// TIA Portal V17 export
// export: Created 2022-06-27T13:58:12.5264541Z, ExportSetting WithDefaults, DisplayName Totally Integrated Automation Portal, DisplayVersion V17 Update 3, DisplayName TIA Portal Openness, DisplayVersion V17 Update 3, DisplayName TIA Portal Version Control Interface, DisplayVersion V17, DisplayName SINAMICS Startdrive Advanced, DisplayVersion V17 Update1, DisplayName SINAMICS Startdrive G110M, G120, G120C, G120D, G120P, G115D, DisplayVersion V17 Update1, DisplayName SINAMICS Startdrive G130, G150, S120, S150, SINAMICS MV, S210, DisplayVersion V17 Update1, DisplayName STEP 7 Professional, DisplayVersion V17 Update 3, DisplayName STEP 7 Safety, DisplayVersion V17, DisplayName WinCC UA Professional, DisplayVersion V17 Update 3
FUNCTION_BLOCK "S05_ANALOGIC_INPUTS"   // FB5, LAD
{ S7_Optimized_Access := 'TRUE' }
VERSION : 0.1
// stored: AutoNumber false, IsIECCheckEnabled false, IsRetainMemResEnabled false, MemoryReserve 100, SetENOAutomatically false, UDAEnableTagReadback false
   VAR
      FB_ANALOGIC_INPUTS_TT82_2E { S7_SetPoint := 'True'} : "FB_ANALOGIC_INPUTS";
      FB_ANALOGIC_INPUTS_TT82_4E { S7_SetPoint := 'True'} : "FB_ANALOGIC_INPUTS";
      FB_ANALOGIC_INPUTS_TT82_6E { S7_SetPoint := 'True'} : "FB_ANALOGIC_INPUTS";
      FB_ANALOGIC_INPUTS_TT82_8E { S7_SetPoint := 'True'} : "FB_ANALOGIC_INPUTS";
      FB_ANALOGIC_INPUTS_TT83_2E { S7_SetPoint := 'True'} : "FB_ANALOGIC_INPUTS";
      FB_ANALOGIC_INPUTS_TT83_4E { S7_SetPoint := 'True'} : "FB_ANALOGIC_INPUTS";
      FB_ANALOGIC_INPUTS_TT83_6E { S7_SetPoint := 'True'} : "FB_ANALOGIC_INPUTS";
      FB_ANALOGIC_INPUTS_TT88_2E { S7_SetPoint := 'True'} : "FB_ANALOGIC_INPUTS";
      FB_ANALOGIC_INPUTS_TT83_8E { S7_SetPoint := 'True'} : "FB_ANALOGIC_INPUTS";
      FB_ANALOGIC_INPUTS_TT84_4E { S7_SetPoint := 'True'} : "FB_ANALOGIC_INPUTS";
      FB_ANALOGIC_INPUTS_TT84_6E { S7_SetPoint := 'True'} : "FB_ANALOGIC_INPUTS";
      FB_ANALOGIC_INPUTS_TT84_8E { S7_SetPoint := 'True'} : "FB_ANALOGIC_INPUTS";
      FB_ANALOGIC_INPUTS_TT85_2E { S7_SetPoint := 'True'} : "FB_ANALOGIC_INPUTS";
   END_VAR
BEGIN

REGION Network 1: TT82-2E - Furnace Thermocouple
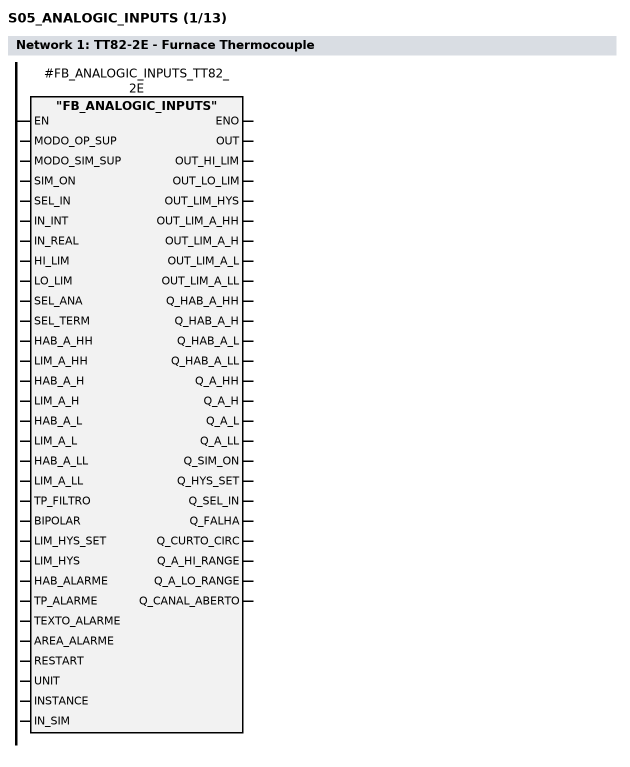
   RUNG wire#powerrail
      #FB_ANALOGIC_INPUTS_TT82_2E(MODO_OP_SUP :=, MODO_SIM_SUP :=, SIM_ON :=, SEL_IN :=, IN_INT :=, IN_REAL :=, HI_LIM :=, LO_LIM :=, SEL_ANA :=, SEL_TERM :=, HAB_A_HH :=, LIM_A_HH :=, HAB_A_H :=, LIM_A_H :=, HAB_A_L :=, LIM_A_L :=, HAB_A_LL :=, LIM_A_LL :=, TP_FILTRO :=, BIPOLAR :=, LIM_HYS_SET :=, LIM_HYS :=, HAB_ALARME :=, TP_ALARME :=, TEXTO_ALARME :=, AREA_ALARME :=, RESTART :=, UNIT :=, INSTANCE :=, IN_SIM :=, OUT =>, OUT_HI_LIM =>, OUT_LO_LIM =>, OUT_LIM_HYS =>, OUT_LIM_A_HH =>, OUT_LIM_A_H =>, OUT_LIM_A_L =>, OUT_LIM_A_LL =>, Q_HAB_A_HH =>, Q_HAB_A_H =>, Q_HAB_A_L =>, Q_HAB_A_LL =>, Q_A_HH =>, Q_A_H =>, Q_A_L =>, Q_A_LL =>, Q_SIM_ON =>, Q_HYS_SET =>, Q_SEL_IN =>, Q_FALHA =>, Q_CURTO_CIRC =>, Q_A_HI_RANGE =>, Q_A_LO_RANGE =>, Q_CANAL_ABERTO =>)
   END_RUNG
   // the same network as SCL:
   #FB_ANALOGIC_INPUTS_TT82_2E();   // "FB_ANALOGIC_INPUTS"
END_REGION

REGION Network 3: TT82-4E - Chamber 1 Air Intake Thermocouple
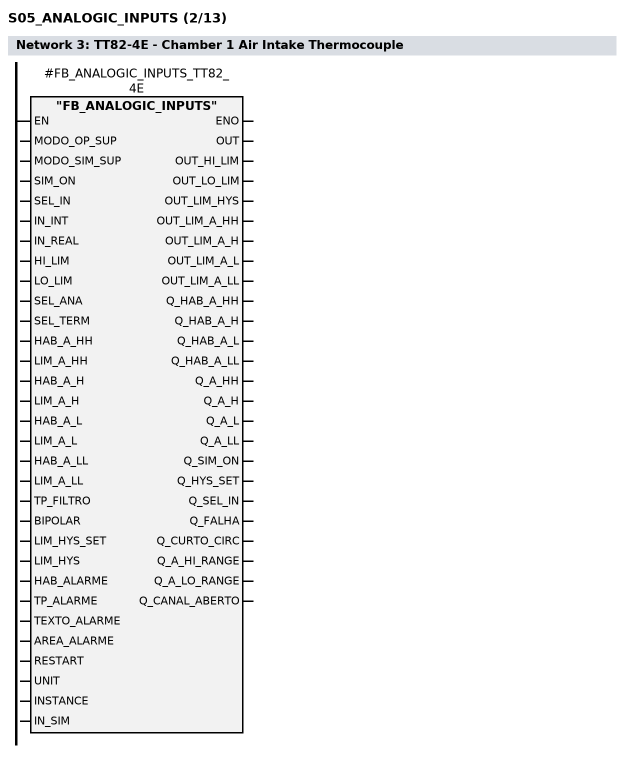
   RUNG wire#powerrail
      #FB_ANALOGIC_INPUTS_TT82_4E(MODO_OP_SUP :=, MODO_SIM_SUP :=, SIM_ON :=, SEL_IN :=, IN_INT :=, IN_REAL :=, HI_LIM :=, LO_LIM :=, SEL_ANA :=, SEL_TERM :=, HAB_A_HH :=, LIM_A_HH :=, HAB_A_H :=, LIM_A_H :=, HAB_A_L :=, LIM_A_L :=, HAB_A_LL :=, LIM_A_LL :=, TP_FILTRO :=, BIPOLAR :=, LIM_HYS_SET :=, LIM_HYS :=, HAB_ALARME :=, TP_ALARME :=, TEXTO_ALARME :=, AREA_ALARME :=, RESTART :=, UNIT :=, INSTANCE :=, IN_SIM :=, OUT =>, OUT_HI_LIM =>, OUT_LO_LIM =>, OUT_LIM_HYS =>, OUT_LIM_A_HH =>, OUT_LIM_A_H =>, OUT_LIM_A_L =>, OUT_LIM_A_LL =>, Q_HAB_A_HH =>, Q_HAB_A_H =>, Q_HAB_A_L =>, Q_HAB_A_LL =>, Q_A_HH =>, Q_A_H =>, Q_A_L =>, Q_A_LL =>, Q_SIM_ON =>, Q_HYS_SET =>, Q_SEL_IN =>, Q_FALHA =>, Q_CURTO_CIRC =>, Q_A_HI_RANGE =>, Q_A_LO_RANGE =>, Q_CANAL_ABERTO =>)
   END_RUNG
   // the same network as SCL:
   #FB_ANALOGIC_INPUTS_TT82_4E();   // "FB_ANALOGIC_INPUTS"
END_REGION

REGION Network 5: TT82-6E - Chamber 2 Air Intake Thermocouple
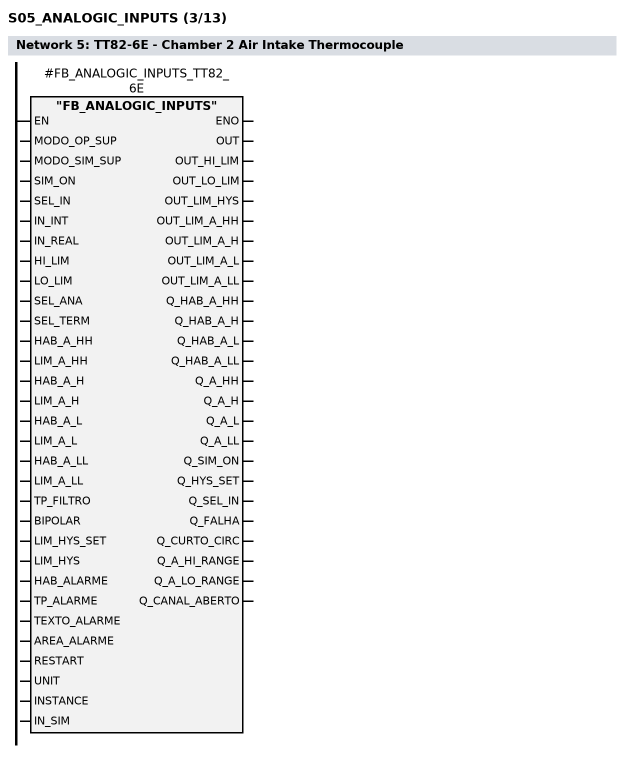
   RUNG wire#powerrail
      #FB_ANALOGIC_INPUTS_TT82_6E(MODO_OP_SUP :=, MODO_SIM_SUP :=, SIM_ON :=, SEL_IN :=, IN_INT :=, IN_REAL :=, HI_LIM :=, LO_LIM :=, SEL_ANA :=, SEL_TERM :=, HAB_A_HH :=, LIM_A_HH :=, HAB_A_H :=, LIM_A_H :=, HAB_A_L :=, LIM_A_L :=, HAB_A_LL :=, LIM_A_LL :=, TP_FILTRO :=, BIPOLAR :=, LIM_HYS_SET :=, LIM_HYS :=, HAB_ALARME :=, TP_ALARME :=, TEXTO_ALARME :=, AREA_ALARME :=, RESTART :=, UNIT :=, INSTANCE :=, IN_SIM :=, OUT =>, OUT_HI_LIM =>, OUT_LO_LIM =>, OUT_LIM_HYS =>, OUT_LIM_A_HH =>, OUT_LIM_A_H =>, OUT_LIM_A_L =>, OUT_LIM_A_LL =>, Q_HAB_A_HH =>, Q_HAB_A_H =>, Q_HAB_A_L =>, Q_HAB_A_LL =>, Q_A_HH =>, Q_A_H =>, Q_A_L =>, Q_A_LL =>, Q_SIM_ON =>, Q_HYS_SET =>, Q_SEL_IN =>, Q_FALHA =>, Q_CURTO_CIRC =>, Q_A_HI_RANGE =>, Q_A_LO_RANGE =>, Q_CANAL_ABERTO =>)
   END_RUNG
   // the same network as SCL:
   #FB_ANALOGIC_INPUTS_TT82_6E();   // "FB_ANALOGIC_INPUTS"
END_REGION

REGION Network 7: TT82-8E - Roaster Air Outtake Thermocouple
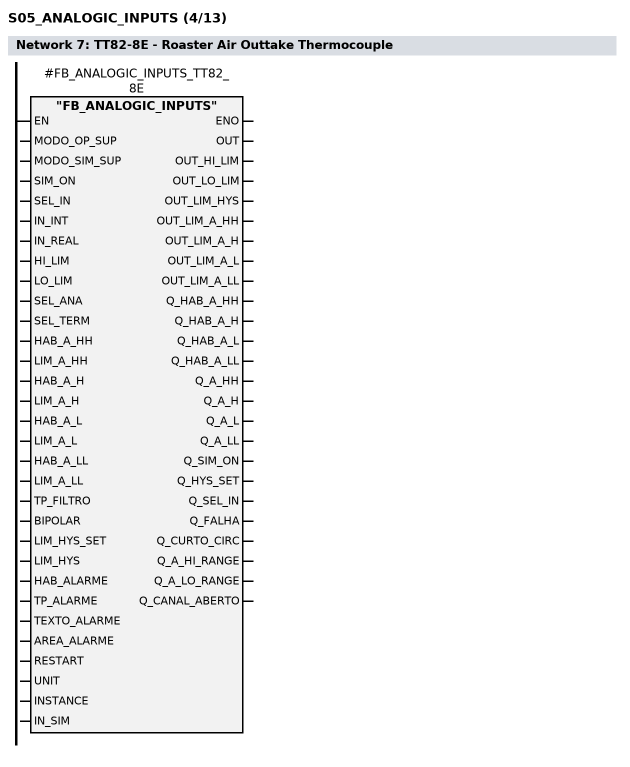
   RUNG wire#powerrail
      #FB_ANALOGIC_INPUTS_TT82_8E(MODO_OP_SUP :=, MODO_SIM_SUP :=, SIM_ON :=, SEL_IN :=, IN_INT :=, IN_REAL :=, HI_LIM :=, LO_LIM :=, SEL_ANA :=, SEL_TERM :=, HAB_A_HH :=, LIM_A_HH :=, HAB_A_H :=, LIM_A_H :=, HAB_A_L :=, LIM_A_L :=, HAB_A_LL :=, LIM_A_LL :=, TP_FILTRO :=, BIPOLAR :=, LIM_HYS_SET :=, LIM_HYS :=, HAB_ALARME :=, TP_ALARME :=, TEXTO_ALARME :=, AREA_ALARME :=, RESTART :=, UNIT :=, INSTANCE :=, IN_SIM :=, OUT =>, OUT_HI_LIM =>, OUT_LO_LIM =>, OUT_LIM_HYS =>, OUT_LIM_A_HH =>, OUT_LIM_A_H =>, OUT_LIM_A_L =>, OUT_LIM_A_LL =>, Q_HAB_A_HH =>, Q_HAB_A_H =>, Q_HAB_A_L =>, Q_HAB_A_LL =>, Q_A_HH =>, Q_A_H =>, Q_A_L =>, Q_A_LL =>, Q_SIM_ON =>, Q_HYS_SET =>, Q_SEL_IN =>, Q_FALHA =>, Q_CURTO_CIRC =>, Q_A_HI_RANGE =>, Q_A_LO_RANGE =>, Q_CANAL_ABERTO =>)
   END_RUNG
   // the same network as SCL:
   #FB_ANALOGIC_INPUTS_TT82_8E();   // "FB_ANALOGIC_INPUTS"
END_REGION

REGION Network 9: TT83-2E - Roaster Cyclone Thermocouple 1
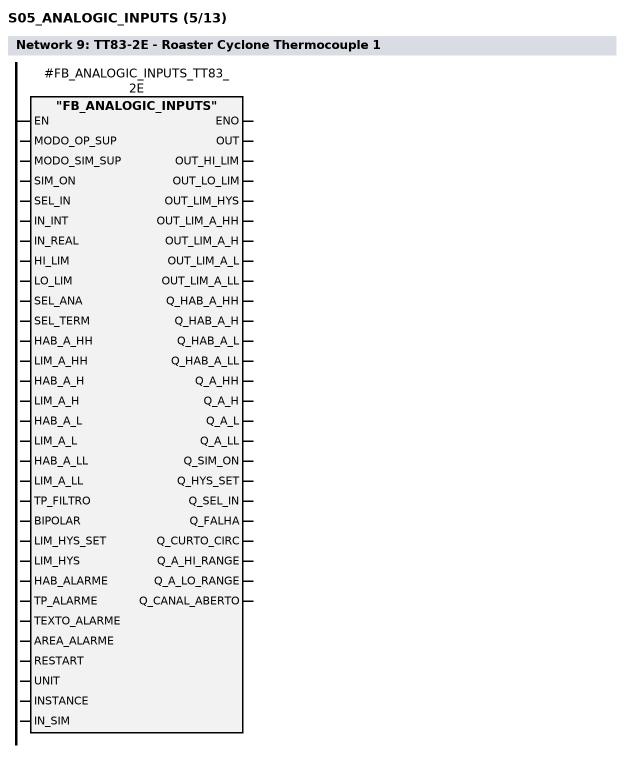
   RUNG wire#powerrail
      #FB_ANALOGIC_INPUTS_TT83_2E(MODO_OP_SUP :=, MODO_SIM_SUP :=, SIM_ON :=, SEL_IN :=, IN_INT :=, IN_REAL :=, HI_LIM :=, LO_LIM :=, SEL_ANA :=, SEL_TERM :=, HAB_A_HH :=, LIM_A_HH :=, HAB_A_H :=, LIM_A_H :=, HAB_A_L :=, LIM_A_L :=, HAB_A_LL :=, LIM_A_LL :=, TP_FILTRO :=, BIPOLAR :=, LIM_HYS_SET :=, LIM_HYS :=, HAB_ALARME :=, TP_ALARME :=, TEXTO_ALARME :=, AREA_ALARME :=, RESTART :=, UNIT :=, INSTANCE :=, IN_SIM :=, OUT =>, OUT_HI_LIM =>, OUT_LO_LIM =>, OUT_LIM_HYS =>, OUT_LIM_A_HH =>, OUT_LIM_A_H =>, OUT_LIM_A_L =>, OUT_LIM_A_LL =>, Q_HAB_A_HH =>, Q_HAB_A_H =>, Q_HAB_A_L =>, Q_HAB_A_LL =>, Q_A_HH =>, Q_A_H =>, Q_A_L =>, Q_A_LL =>, Q_SIM_ON =>, Q_HYS_SET =>, Q_SEL_IN =>, Q_FALHA =>, Q_CURTO_CIRC =>, Q_A_HI_RANGE =>, Q_A_LO_RANGE =>, Q_CANAL_ABERTO =>)
   END_RUNG
   // the same network as SCL:
   #FB_ANALOGIC_INPUTS_TT83_2E();   // "FB_ANALOGIC_INPUTS"
END_REGION

REGION Network 11: TT83-4E - Roaster Cyclone Thermocouple 2
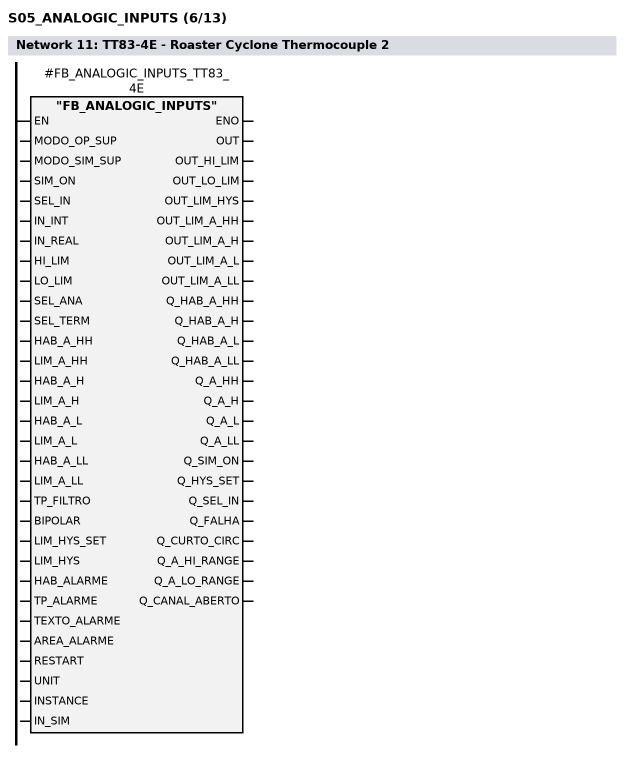
   RUNG wire#powerrail
      #FB_ANALOGIC_INPUTS_TT83_4E(MODO_OP_SUP :=, MODO_SIM_SUP :=, SIM_ON :=, SEL_IN :=, IN_INT :=, IN_REAL :=, HI_LIM :=, LO_LIM :=, SEL_ANA :=, SEL_TERM :=, HAB_A_HH :=, LIM_A_HH :=, HAB_A_H :=, LIM_A_H :=, HAB_A_L :=, LIM_A_L :=, HAB_A_LL :=, LIM_A_LL :=, TP_FILTRO :=, BIPOLAR :=, LIM_HYS_SET :=, LIM_HYS :=, HAB_ALARME :=, TP_ALARME :=, TEXTO_ALARME :=, AREA_ALARME :=, RESTART :=, UNIT :=, INSTANCE :=, IN_SIM :=, OUT =>, OUT_HI_LIM =>, OUT_LO_LIM =>, OUT_LIM_HYS =>, OUT_LIM_A_HH =>, OUT_LIM_A_H =>, OUT_LIM_A_L =>, OUT_LIM_A_LL =>, Q_HAB_A_HH =>, Q_HAB_A_H =>, Q_HAB_A_L =>, Q_HAB_A_LL =>, Q_A_HH =>, Q_A_H =>, Q_A_L =>, Q_A_LL =>, Q_SIM_ON =>, Q_HYS_SET =>, Q_SEL_IN =>, Q_FALHA =>, Q_CURTO_CIRC =>, Q_A_HI_RANGE =>, Q_A_LO_RANGE =>, Q_CANAL_ABERTO =>)
   END_RUNG
   // the same network as SCL:
   #FB_ANALOGIC_INPUTS_TT83_4E();   // "FB_ANALOGIC_INPUTS"
END_REGION

REGION Network 13: TT83-6E - Chamber 1 Thermocouple 1
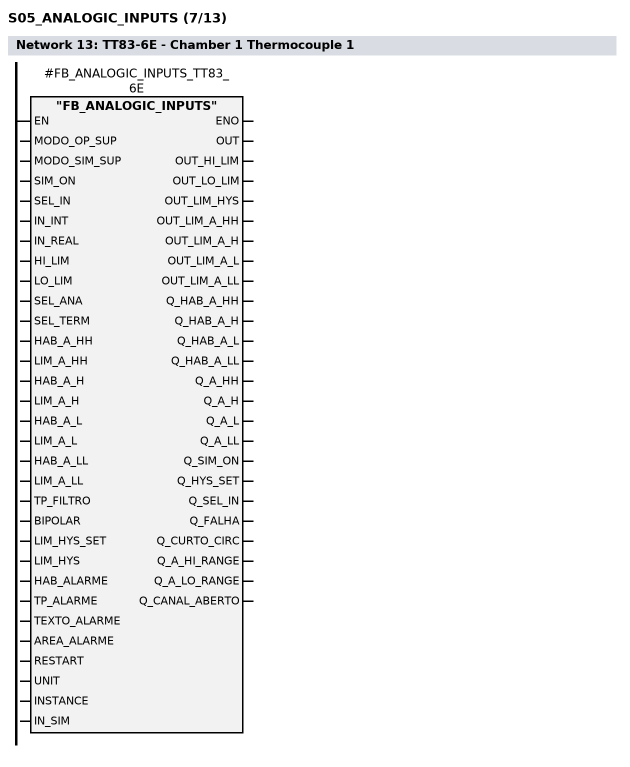
   RUNG wire#powerrail
      #FB_ANALOGIC_INPUTS_TT83_6E(MODO_OP_SUP :=, MODO_SIM_SUP :=, SIM_ON :=, SEL_IN :=, IN_INT :=, IN_REAL :=, HI_LIM :=, LO_LIM :=, SEL_ANA :=, SEL_TERM :=, HAB_A_HH :=, LIM_A_HH :=, HAB_A_H :=, LIM_A_H :=, HAB_A_L :=, LIM_A_L :=, HAB_A_LL :=, LIM_A_LL :=, TP_FILTRO :=, BIPOLAR :=, LIM_HYS_SET :=, LIM_HYS :=, HAB_ALARME :=, TP_ALARME :=, TEXTO_ALARME :=, AREA_ALARME :=, RESTART :=, UNIT :=, INSTANCE :=, IN_SIM :=, OUT =>, OUT_HI_LIM =>, OUT_LO_LIM =>, OUT_LIM_HYS =>, OUT_LIM_A_HH =>, OUT_LIM_A_H =>, OUT_LIM_A_L =>, OUT_LIM_A_LL =>, Q_HAB_A_HH =>, Q_HAB_A_H =>, Q_HAB_A_L =>, Q_HAB_A_LL =>, Q_A_HH =>, Q_A_H =>, Q_A_L =>, Q_A_LL =>, Q_SIM_ON =>, Q_HYS_SET =>, Q_SEL_IN =>, Q_FALHA =>, Q_CURTO_CIRC =>, Q_A_HI_RANGE =>, Q_A_LO_RANGE =>, Q_CANAL_ABERTO =>)
   END_RUNG
   // the same network as SCL:
   #FB_ANALOGIC_INPUTS_TT83_6E();   // "FB_ANALOGIC_INPUTS"
END_REGION

REGION Network 15: TT88-2E - Chamber 1 Thermocouple 2
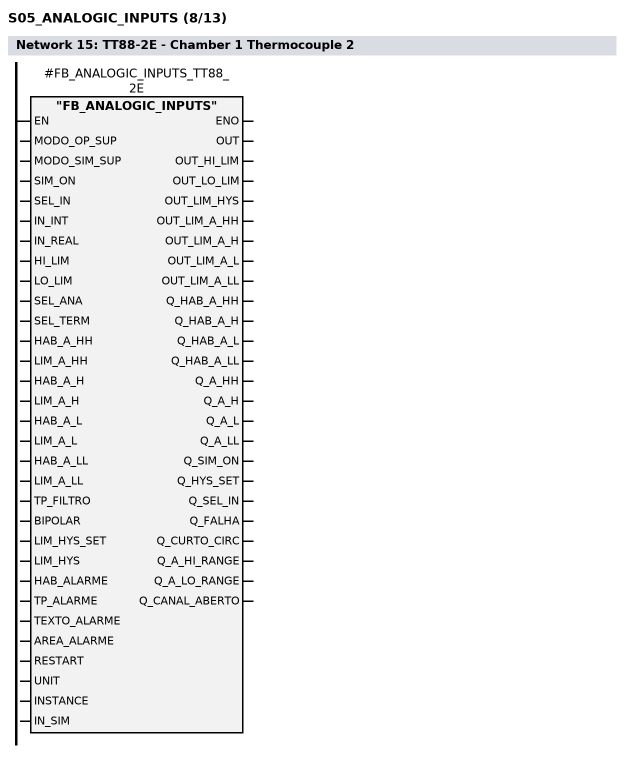
   RUNG wire#powerrail
      #FB_ANALOGIC_INPUTS_TT88_2E(MODO_OP_SUP :=, MODO_SIM_SUP :=, SIM_ON :=, SEL_IN :=, IN_INT :=, IN_REAL :=, HI_LIM :=, LO_LIM :=, SEL_ANA :=, SEL_TERM :=, HAB_A_HH :=, LIM_A_HH :=, HAB_A_H :=, LIM_A_H :=, HAB_A_L :=, LIM_A_L :=, HAB_A_LL :=, LIM_A_LL :=, TP_FILTRO :=, BIPOLAR :=, LIM_HYS_SET :=, LIM_HYS :=, HAB_ALARME :=, TP_ALARME :=, TEXTO_ALARME :=, AREA_ALARME :=, RESTART :=, UNIT :=, INSTANCE :=, IN_SIM :=, OUT =>, OUT_HI_LIM =>, OUT_LO_LIM =>, OUT_LIM_HYS =>, OUT_LIM_A_HH =>, OUT_LIM_A_H =>, OUT_LIM_A_L =>, OUT_LIM_A_LL =>, Q_HAB_A_HH =>, Q_HAB_A_H =>, Q_HAB_A_L =>, Q_HAB_A_LL =>, Q_A_HH =>, Q_A_H =>, Q_A_L =>, Q_A_LL =>, Q_SIM_ON =>, Q_HYS_SET =>, Q_SEL_IN =>, Q_FALHA =>, Q_CURTO_CIRC =>, Q_A_HI_RANGE =>, Q_A_LO_RANGE =>, Q_CANAL_ABERTO =>)
   END_RUNG
   // the same network as SCL:
   #FB_ANALOGIC_INPUTS_TT88_2E();   // "FB_ANALOGIC_INPUTS"
END_REGION

REGION Network 17: TT83-8E - Chamber 2 Thermocouple 1
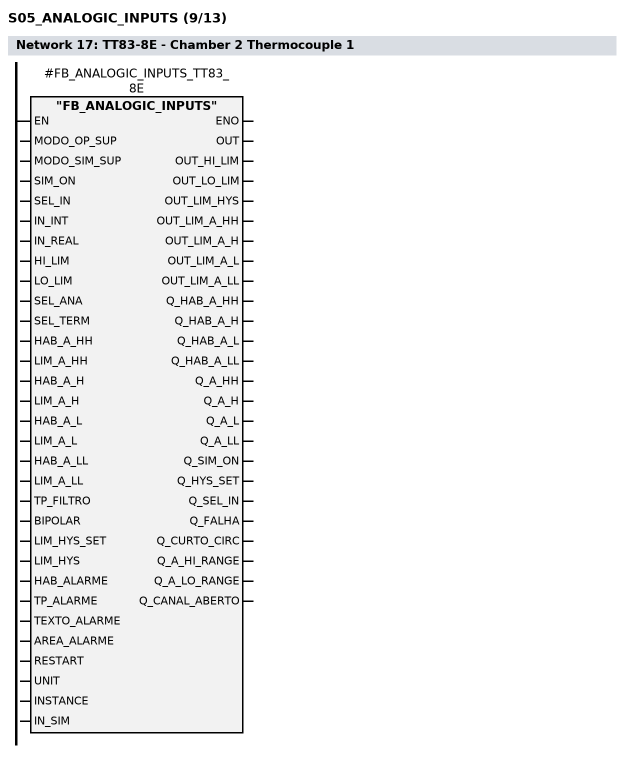
   RUNG wire#powerrail
      #FB_ANALOGIC_INPUTS_TT83_8E(MODO_OP_SUP :=, MODO_SIM_SUP :=, SIM_ON :=, SEL_IN :=, IN_INT :=, IN_REAL :=, HI_LIM :=, LO_LIM :=, SEL_ANA :=, SEL_TERM :=, HAB_A_HH :=, LIM_A_HH :=, HAB_A_H :=, LIM_A_H :=, HAB_A_L :=, LIM_A_L :=, HAB_A_LL :=, LIM_A_LL :=, TP_FILTRO :=, BIPOLAR :=, LIM_HYS_SET :=, LIM_HYS :=, HAB_ALARME :=, TP_ALARME :=, TEXTO_ALARME :=, AREA_ALARME :=, RESTART :=, UNIT :=, INSTANCE :=, IN_SIM :=, OUT =>, OUT_HI_LIM =>, OUT_LO_LIM =>, OUT_LIM_HYS =>, OUT_LIM_A_HH =>, OUT_LIM_A_H =>, OUT_LIM_A_L =>, OUT_LIM_A_LL =>, Q_HAB_A_HH =>, Q_HAB_A_H =>, Q_HAB_A_L =>, Q_HAB_A_LL =>, Q_A_HH =>, Q_A_H =>, Q_A_L =>, Q_A_LL =>, Q_SIM_ON =>, Q_HYS_SET =>, Q_SEL_IN =>, Q_FALHA =>, Q_CURTO_CIRC =>, Q_A_HI_RANGE =>, Q_A_LO_RANGE =>, Q_CANAL_ABERTO =>)
   END_RUNG
   // the same network as SCL:
   #FB_ANALOGIC_INPUTS_TT83_8E();   // "FB_ANALOGIC_INPUTS"
END_REGION

REGION Network 19: TT84-4E - Chamber 2 Thermocouple 2
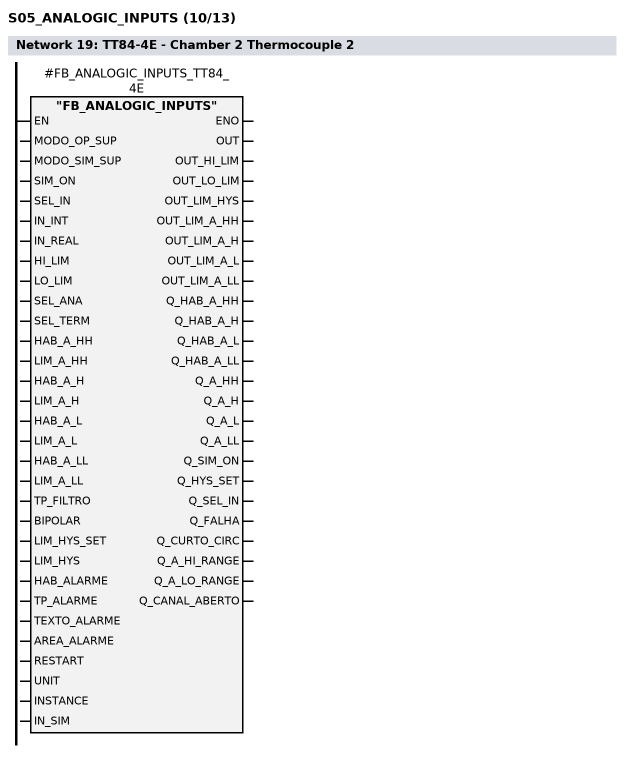
   RUNG wire#powerrail
      #FB_ANALOGIC_INPUTS_TT84_4E(MODO_OP_SUP :=, MODO_SIM_SUP :=, SIM_ON :=, SEL_IN :=, IN_INT :=, IN_REAL :=, HI_LIM :=, LO_LIM :=, SEL_ANA :=, SEL_TERM :=, HAB_A_HH :=, LIM_A_HH :=, HAB_A_H :=, LIM_A_H :=, HAB_A_L :=, LIM_A_L :=, HAB_A_LL :=, LIM_A_LL :=, TP_FILTRO :=, BIPOLAR :=, LIM_HYS_SET :=, LIM_HYS :=, HAB_ALARME :=, TP_ALARME :=, TEXTO_ALARME :=, AREA_ALARME :=, RESTART :=, UNIT :=, INSTANCE :=, IN_SIM :=, OUT =>, OUT_HI_LIM =>, OUT_LO_LIM =>, OUT_LIM_HYS =>, OUT_LIM_A_HH =>, OUT_LIM_A_H =>, OUT_LIM_A_L =>, OUT_LIM_A_LL =>, Q_HAB_A_HH =>, Q_HAB_A_H =>, Q_HAB_A_L =>, Q_HAB_A_LL =>, Q_A_HH =>, Q_A_H =>, Q_A_L =>, Q_A_LL =>, Q_SIM_ON =>, Q_HYS_SET =>, Q_SEL_IN =>, Q_FALHA =>, Q_CURTO_CIRC =>, Q_A_HI_RANGE =>, Q_A_LO_RANGE =>, Q_CANAL_ABERTO =>)
   END_RUNG
   // the same network as SCL:
   #FB_ANALOGIC_INPUTS_TT84_4E();   // "FB_ANALOGIC_INPUTS"
END_REGION

REGION Network 21: TT84-6E - Cooler 1 Thermocouple
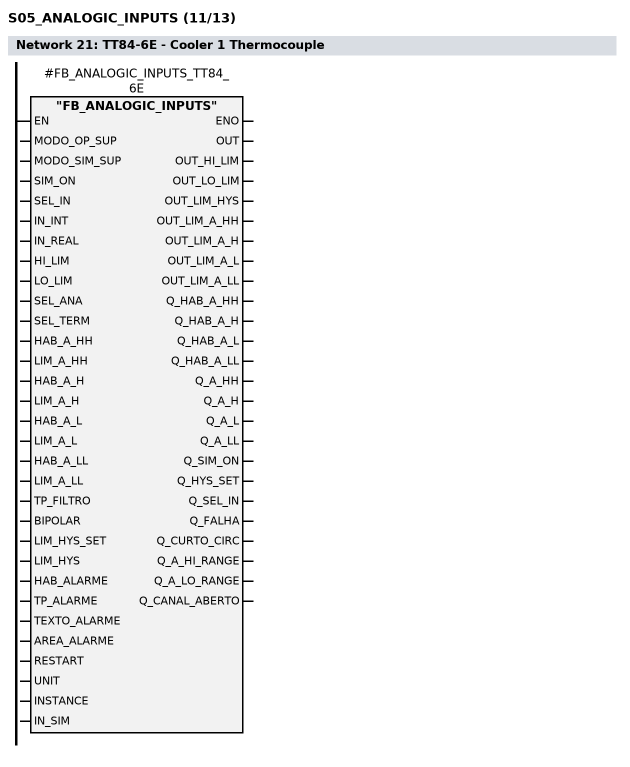
   RUNG wire#powerrail
      #FB_ANALOGIC_INPUTS_TT84_6E(MODO_OP_SUP :=, MODO_SIM_SUP :=, SIM_ON :=, SEL_IN :=, IN_INT :=, IN_REAL :=, HI_LIM :=, LO_LIM :=, SEL_ANA :=, SEL_TERM :=, HAB_A_HH :=, LIM_A_HH :=, HAB_A_H :=, LIM_A_H :=, HAB_A_L :=, LIM_A_L :=, HAB_A_LL :=, LIM_A_LL :=, TP_FILTRO :=, BIPOLAR :=, LIM_HYS_SET :=, LIM_HYS :=, HAB_ALARME :=, TP_ALARME :=, TEXTO_ALARME :=, AREA_ALARME :=, RESTART :=, UNIT :=, INSTANCE :=, IN_SIM :=, OUT =>, OUT_HI_LIM =>, OUT_LO_LIM =>, OUT_LIM_HYS =>, OUT_LIM_A_HH =>, OUT_LIM_A_H =>, OUT_LIM_A_L =>, OUT_LIM_A_LL =>, Q_HAB_A_HH =>, Q_HAB_A_H =>, Q_HAB_A_L =>, Q_HAB_A_LL =>, Q_A_HH =>, Q_A_H =>, Q_A_L =>, Q_A_LL =>, Q_SIM_ON =>, Q_HYS_SET =>, Q_SEL_IN =>, Q_FALHA =>, Q_CURTO_CIRC =>, Q_A_HI_RANGE =>, Q_A_LO_RANGE =>, Q_CANAL_ABERTO =>)
   END_RUNG
   // the same network as SCL:
   #FB_ANALOGIC_INPUTS_TT84_6E();   // "FB_ANALOGIC_INPUTS"
END_REGION

REGION Network 23: TT84-8E - Cooler 2 Thermocouple
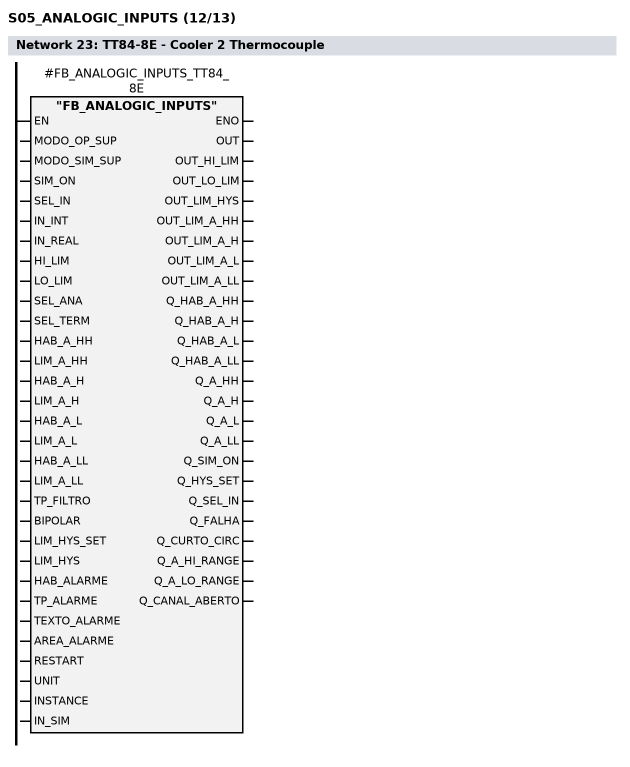
   RUNG wire#powerrail
      #FB_ANALOGIC_INPUTS_TT84_8E(MODO_OP_SUP :=, MODO_SIM_SUP :=, SIM_ON :=, SEL_IN :=, IN_INT :=, IN_REAL :=, HI_LIM :=, LO_LIM :=, SEL_ANA :=, SEL_TERM :=, HAB_A_HH :=, LIM_A_HH :=, HAB_A_H :=, LIM_A_H :=, HAB_A_L :=, LIM_A_L :=, HAB_A_LL :=, LIM_A_LL :=, TP_FILTRO :=, BIPOLAR :=, LIM_HYS_SET :=, LIM_HYS :=, HAB_ALARME :=, TP_ALARME :=, TEXTO_ALARME :=, AREA_ALARME :=, RESTART :=, UNIT :=, INSTANCE :=, IN_SIM :=, OUT =>, OUT_HI_LIM =>, OUT_LO_LIM =>, OUT_LIM_HYS =>, OUT_LIM_A_HH =>, OUT_LIM_A_H =>, OUT_LIM_A_L =>, OUT_LIM_A_LL =>, Q_HAB_A_HH =>, Q_HAB_A_H =>, Q_HAB_A_L =>, Q_HAB_A_LL =>, Q_A_HH =>, Q_A_H =>, Q_A_L =>, Q_A_LL =>, Q_SIM_ON =>, Q_HYS_SET =>, Q_SEL_IN =>, Q_FALHA =>, Q_CURTO_CIRC =>, Q_A_HI_RANGE =>, Q_A_LO_RANGE =>, Q_CANAL_ABERTO =>)
   END_RUNG
   // the same network as SCL:
   #FB_ANALOGIC_INPUTS_TT84_8E();   // "FB_ANALOGIC_INPUTS"
END_REGION

REGION Network 25: TT85-2E - Smoke Thermocouple
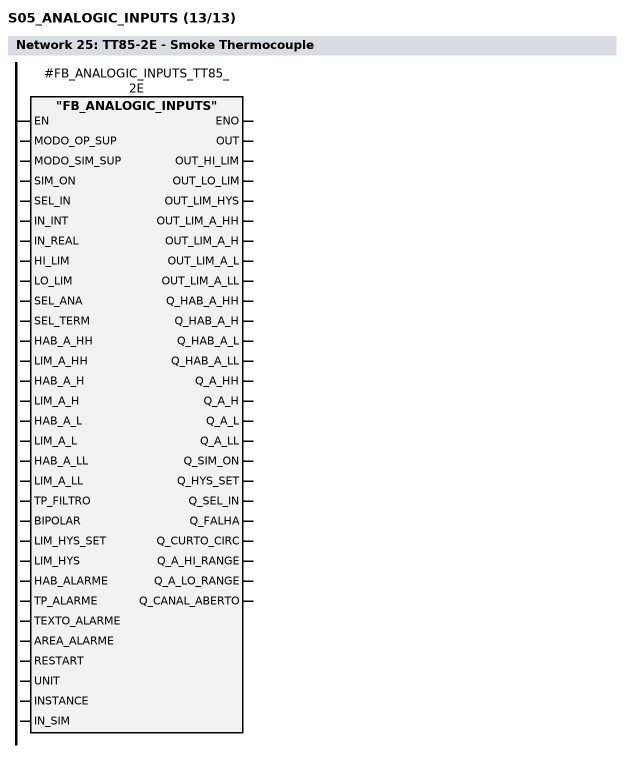
   RUNG wire#powerrail
      #FB_ANALOGIC_INPUTS_TT85_2E(MODO_OP_SUP :=, MODO_SIM_SUP :=, SIM_ON :=, SEL_IN :=, IN_INT :=, IN_REAL :=, HI_LIM :=, LO_LIM :=, SEL_ANA :=, SEL_TERM :=, HAB_A_HH :=, LIM_A_HH :=, HAB_A_H :=, LIM_A_H :=, HAB_A_L :=, LIM_A_L :=, HAB_A_LL :=, LIM_A_LL :=, TP_FILTRO :=, BIPOLAR :=, LIM_HYS_SET :=, LIM_HYS :=, HAB_ALARME :=, TP_ALARME :=, TEXTO_ALARME :=, AREA_ALARME :=, RESTART :=, UNIT :=, INSTANCE :=, IN_SIM :=, OUT =>, OUT_HI_LIM =>, OUT_LO_LIM =>, OUT_LIM_HYS =>, OUT_LIM_A_HH =>, OUT_LIM_A_H =>, OUT_LIM_A_L =>, OUT_LIM_A_LL =>, Q_HAB_A_HH =>, Q_HAB_A_H =>, Q_HAB_A_L =>, Q_HAB_A_LL =>, Q_A_HH =>, Q_A_H =>, Q_A_L =>, Q_A_LL =>, Q_SIM_ON =>, Q_HYS_SET =>, Q_SEL_IN =>, Q_FALHA =>, Q_CURTO_CIRC =>, Q_A_HI_RANGE =>, Q_A_LO_RANGE =>, Q_CANAL_ABERTO =>)
   END_RUNG
   // the same network as SCL:
   #FB_ANALOGIC_INPUTS_TT85_2E();   // "FB_ANALOGIC_INPUTS"
END_REGION

REGION Network 27: VR88-2E - Rear Bearing Vibration Sensor - Roaster Fan
END_REGION

REGION Network 29: VR88-4E - Front Bearing Vibration Sensor - Roaster Fan
END_REGION

REGION Network 31: VR88-6E - Rear Bearing Vibration Sensor - Dryer Fan
END_REGION

REGION Network 33: VR88-8E - Front Bearing Vibration Sensor - Dryer Fan
END_REGION

REGION Network 35: BCV99-2B - Burner Speed Setpoint
END_REGION
END_FUNCTION_BLOCK
